FUNCTION_BLOCK WinlineUXR100040G IMPLEMENTS ACDCChargerElement
VAR_INPUT
END_VAR

VAR_OUTPUT
END_VAR

VAR
	
END_VAR


VAR CONSTANT
	UnitPower	:	Real := 40;
END_VAR

METHOD Disable : BOOL
VAR_INPUT
END_VAR
END_METHOD

METHOD Enable : BOOL
VAR_INPUT
END_VAR
END_METHOD

METHOD SetPowerLevel : BOOL
VAR_INPUT
END_VAR
END_METHOD

END_FUNCTION_BLOCK

(* stored: Version 1.1.0.1, ProductVersion 3.1.4024.12
   POU WinlineUXR100040G: Id {bcc9d53c-d926-49d7-a9d7-e15bbef623fc}, SpecialFunc None
   Method Disable: Id {6718066a-b33b-4271-b0de-4ea0b20b15bc}
   Method Enable: Id {752dabc4-f475-475c-bbcb-40c8349eda22}
   Method SetPowerLevel: Id {ebd03c02-44b6-4acf-b972-f4a5bc639d09} *)
